{attribute 'qualified_only'}
{attribute 'strict'}
TYPE nTestType :
(
	none := 0,
	testEOL := 10,
	testPerformance := 20,
	testHour := 30,
	testWhole := 40,
	testCyclic30 := 50,
	testCyclic70 := 60
);
END_TYPE

(* stored: Version 1.1.0.1, ProductVersion 3.1.4024.12
   DUT nTestType: Id {f98a8cbd-837e-4708-8668-b582b3550552} *)
